(* CoDeSys 2.3.9.28 project: Automacao_ProjetoSemestral.pro *)
(* Libraries: Standard.lib 27.1.09 11:27:38, Util.lib 27.1.09 11:27:38, IecSfc.lib 24.11.08 08:07:15, SysLibTime.lib 27.1.09 11:27:38, SysTaskInfo.lib 24.11.08 08:07:15, SYSLIBCALLBACK.LIB 27.1.09 11:27:38 *)

(* PLC configuration (modules and I/O channels)
CPX-CEC [Root] node -1, in %IB0 out %QB0 {StringParam = 2773,0,0,0,0; ByteParam = 0; ByteParam = 31; ByteParam = 0; ByteParam = 0; ByteParam = 0; ByteParam = 0; ByteParam = 0; ByteParam = 0; ByteParam = 2; ByteParam = 0; ByteParam = 0; ByteParam = 0; ByteParam = 32; ByteParam = 0; ByteParam = 0; ByteParam = 5; ByteParam = 0; ByteParam = 0; ByteParam = 0; ByteParam = 0; ByteParam = 0; ByteParam = 0; ByteParam = 0; ByteParam = 0; ByteParam = 14; ByteParam = 240; ByteParam = 192; ByteParam = 168; ByteParam = 2; ByteParam = 10; ByteParam = 255; ByteParam = 255; ByteParam = 0; ByteParam = 0; ByteParam = 192; ByteParam = 168; ByteParam = 1; ByteParam = 1; ByteParam = 192; ByteParam = 168; ByteParam = 2; ByteParam = 10; ByteParam = 255; ByteParam = 255; ByteParam = 0; ByteParam = 0; ByteParam = 192; ByteParam = 168; ByteParam = 1; ByteParam = 1}
  Hexswitch AT %IB0 [HexSwitch] rotary switch 0 = STOP, 1-15 = RUN
  IOModules [CPX_MASTER] node 0, in %IB4 out %QB0
*)

(* Global variable list: Global_Variables *)
VAR_GLOBAL

	M1 : BOOL;
	M2 : BOOL;
	P1 : BOOL;
	P2_IDA : BOOL;
	P2_VOLTA : BOOL;
	P3 : BOOL;
	LP_1 : BOOL;
	LP_2 : BOOL;
	AL: BOOL;

	START AT %QX2.0 : BOOL;
	STOP AT %QX2.1 : BOOL;
	S1 AT %QX0.2 : BOOL;
	S2 AT %QX0.3 : BOOL;
	S3 AT %QX0.4 : BOOL;
	S4 AT %QX0.5 : BOOL;
	S5 AT %QX0.6 : BOOL;
	S6 AT %QX0.7 : BOOL;
	S7 AT %QX0.8 : BOOL;

	M_START : BOOL;
	M_CONT: BOOL;
	M_P1: BOOL;
	M_TEMPERA: BOOL;
	M_2_ENT : BOOL;
	M_2_SAI : BOOL;

	MT_1 : BOOL;
	MT_2 : BOOL;
	MT_3 : BOOL;
	MT_4 : BOOL;
	MT_5 : BOOL;

	T_TEMPERA : TON;
	T_P1 : TOF;
	T_ALARME1:TON;
	T_ALARME2:TON;

    CONT_2_ENT: CTU;
	CONT_2_SAI : CTU;

END_VAR

(* POU PLC_PRG, LD *)
PROGRAM PLC_PRG
VAR
END_VAR
VAR (* helpers for the ST form of the networks *)
	_p1 : BOOL;
	_p2 : BOOL;
	_p3 : BOOL;
END_VAR
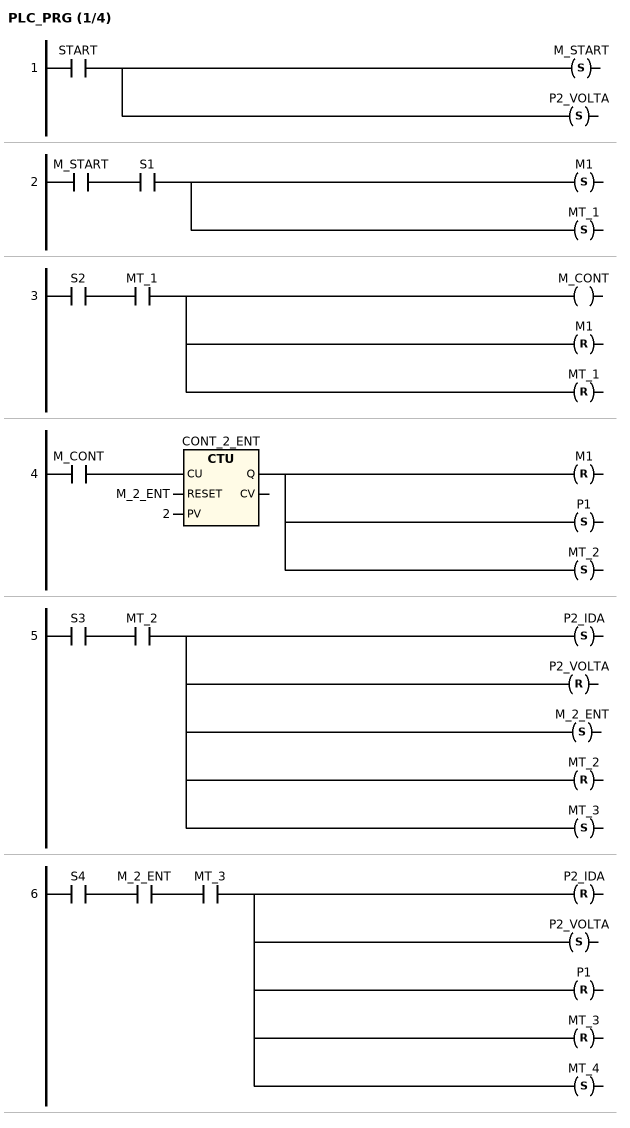
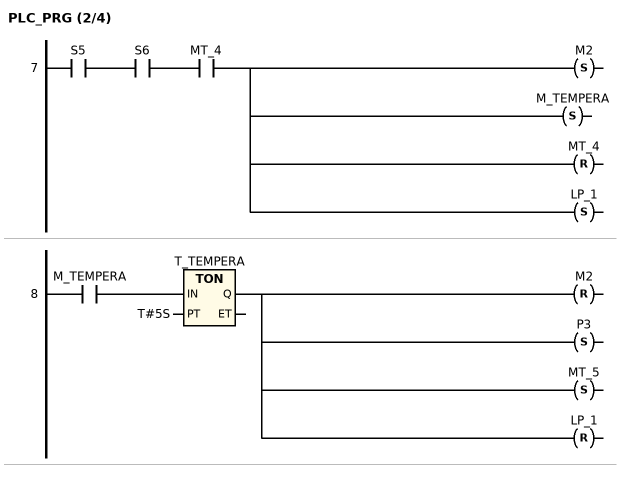
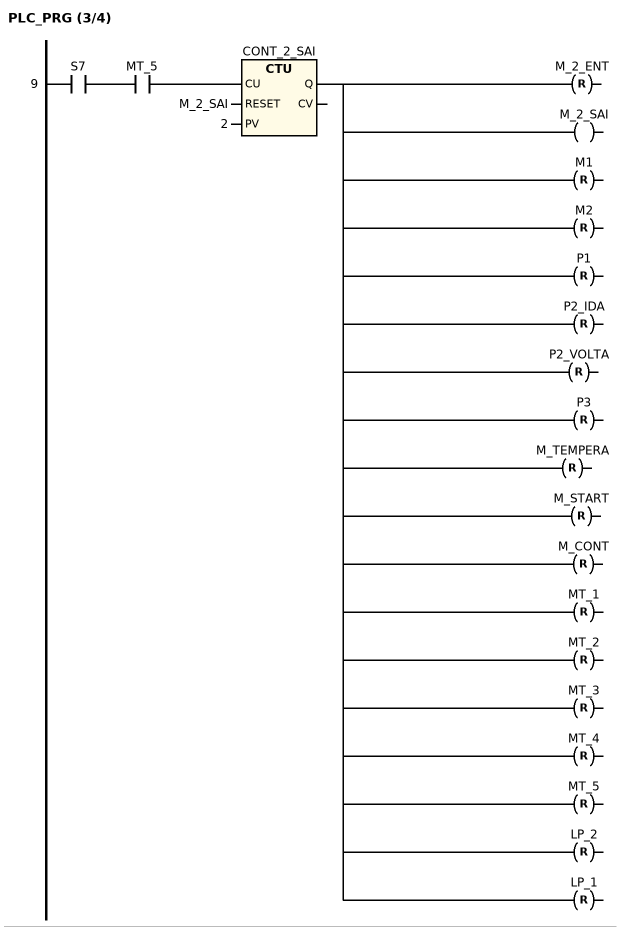
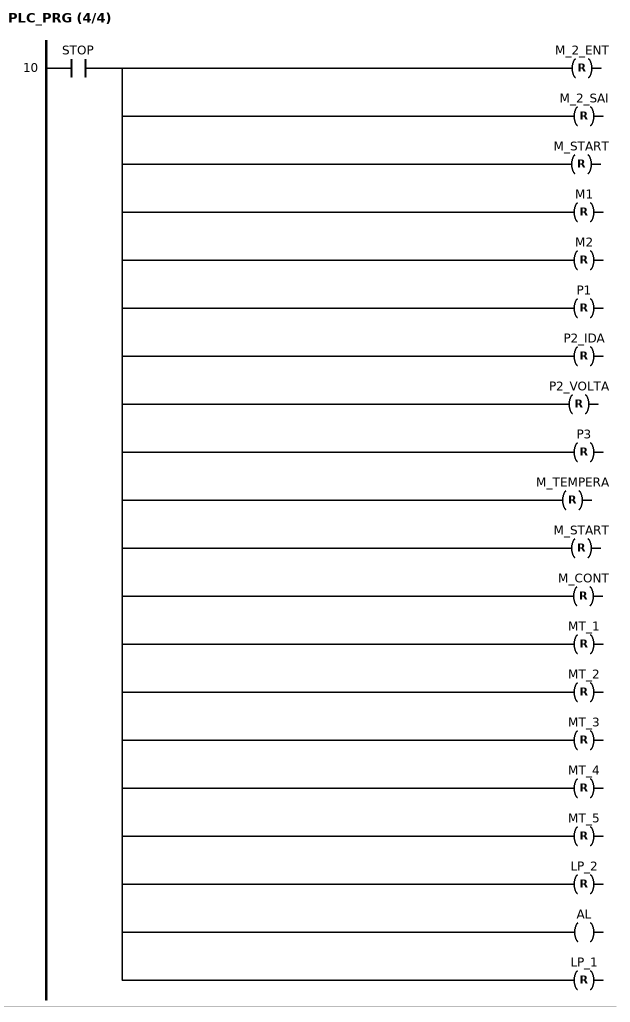
_LD_ (* Ladder Diagram *)
NETWORK 1
	[START] --- (S M_START) (S P2_VOLTA)
NETWORK 2
	[M_START] - [S1] --- (S M1) (S MT_1)
NETWORK 3
	[S2] - [MT_1] --- (M_CONT) (R M1) (R MT_1)
NETWORK 4
	[M_CONT] - CONT_2_ENT:CTU(CU: *, RESET: M_2_ENT, PV: 2) --- (R M1) (S P1) (S MT_2)
NETWORK 5
	[S3] - [MT_2] --- (S P2_IDA) (R P2_VOLTA) (S M_2_ENT) (R MT_2) (S MT_3)
NETWORK 6
	[S4] - [M_2_ENT] - [MT_3] --- (R P2_IDA) (S P2_VOLTA) (R P1) (R MT_3) (S MT_4)
NETWORK 7
	[S5] - [S6] - [MT_4] --- (S M2) (S M_TEMPERA) (R MT_4) (S LP_1)
NETWORK 8
	[M_TEMPERA] - T_TEMPERA:TON(IN: *, PT: T#5S) --- (R M2) (S P3) (S MT_5) (R LP_1)
NETWORK 9
	[S7] - [MT_5] - CONT_2_SAI:CTU(CU: *, RESET: M_2_SAI, PV: 2) --- (R M_2_ENT) (M_2_SAI) (R M1) (R M2) (R P1) (R P2_IDA) (R P2_VOLTA) (R P3) (R M_TEMPERA) (R M_START) (R M_CONT) (R MT_1) (R MT_2) (R MT_3) (R MT_4) (R MT_5) (R LP_2) (R LP_1)
NETWORK 10
	[STOP] --- (R M_2_ENT) (R M_2_SAI) (R M_START) (R M1) (R M2) (R P1) (R P2_IDA) (R P2_VOLTA) (R P3) (R M_TEMPERA) (R M_START) (R M_CONT) (R MT_1) (R MT_2) (R MT_3) (R MT_4) (R MT_5) (R LP_2) (AL) (R LP_1)
_END_LD_
(* the same logic as Structured Text *)
(* Network 1 *)
IF START THEN M_START := TRUE; P2_VOLTA := TRUE; END_IF;
(* Network 2 *)
IF M_START AND S1 THEN M1 := TRUE; MT_1 := TRUE; END_IF;
(* Network 3 *)
M_CONT := S2 AND MT_1;
IF M_CONT THEN M1 := FALSE; MT_1 := FALSE; END_IF;
(* Network 4 *)
CONT_2_ENT(CU := M_CONT, RESET := M_2_ENT, PV := 2);
IF CONT_2_ENT.Q THEN M1 := FALSE; P1 := TRUE; MT_2 := TRUE; END_IF;
(* Network 5 *)
_p1 := S3 AND MT_2;
IF _p1 THEN P2_IDA := TRUE; P2_VOLTA := FALSE; M_2_ENT := TRUE; MT_2 := FALSE; MT_3 := TRUE; END_IF;
(* Network 6 *)
_p2 := S4 AND M_2_ENT AND MT_3;
IF _p2 THEN P2_IDA := FALSE; P2_VOLTA := TRUE; P1 := FALSE; MT_3 := FALSE; MT_4 := TRUE; END_IF;
(* Network 7 *)
_p3 := S5 AND S6 AND MT_4;
IF _p3 THEN M2 := TRUE; M_TEMPERA := TRUE; MT_4 := FALSE; LP_1 := TRUE; END_IF;
(* Network 8 *)
T_TEMPERA(IN := M_TEMPERA, PT := T#5S);
IF T_TEMPERA.Q THEN M2 := FALSE; P3 := TRUE; MT_5 := TRUE; LP_1 := FALSE; END_IF;
(* Network 9 *)
CONT_2_SAI(CU := S7 AND MT_5, RESET := M_2_SAI, PV := 2);
IF CONT_2_SAI.Q THEN M_2_ENT := FALSE; END_IF;
M_2_SAI := CONT_2_SAI.Q;
IF CONT_2_SAI.Q THEN M1 := FALSE; END_IF;
IF CONT_2_SAI.Q THEN M2 := FALSE; END_IF;
IF CONT_2_SAI.Q THEN P1 := FALSE; END_IF;
IF CONT_2_SAI.Q THEN P2_IDA := FALSE; END_IF;
IF CONT_2_SAI.Q THEN P2_VOLTA := FALSE; END_IF;
IF CONT_2_SAI.Q THEN P3 := FALSE; END_IF;
IF CONT_2_SAI.Q THEN M_TEMPERA := FALSE; END_IF;
IF CONT_2_SAI.Q THEN M_START := FALSE; END_IF;
IF CONT_2_SAI.Q THEN M_CONT := FALSE; END_IF;
IF CONT_2_SAI.Q THEN MT_1 := FALSE; END_IF;
IF CONT_2_SAI.Q THEN MT_2 := FALSE; END_IF;
IF CONT_2_SAI.Q THEN MT_3 := FALSE; END_IF;
IF CONT_2_SAI.Q THEN MT_4 := FALSE; END_IF;
IF CONT_2_SAI.Q THEN MT_5 := FALSE; END_IF;
IF CONT_2_SAI.Q THEN LP_2 := FALSE; END_IF;
IF CONT_2_SAI.Q THEN LP_1 := FALSE; END_IF;
(* Network 10 *)
IF STOP THEN M_2_ENT := FALSE; END_IF;
IF STOP THEN M_2_SAI := FALSE; END_IF;
IF STOP THEN M_START := FALSE; END_IF;
IF STOP THEN M1 := FALSE; END_IF;
IF STOP THEN M2 := FALSE; END_IF;
IF STOP THEN P1 := FALSE; END_IF;
IF STOP THEN P2_IDA := FALSE; END_IF;
IF STOP THEN P2_VOLTA := FALSE; END_IF;
IF STOP THEN P3 := FALSE; END_IF;
IF STOP THEN M_TEMPERA := FALSE; END_IF;
IF STOP THEN M_START := FALSE; END_IF;
IF STOP THEN M_CONT := FALSE; END_IF;
IF STOP THEN MT_1 := FALSE; END_IF;
IF STOP THEN MT_2 := FALSE; END_IF;
IF STOP THEN MT_3 := FALSE; END_IF;
IF STOP THEN MT_4 := FALSE; END_IF;
IF STOP THEN MT_5 := FALSE; END_IF;
IF STOP THEN LP_2 := FALSE; END_IF;
AL := STOP;
IF STOP THEN LP_1 := FALSE; END_IF;
END_PROGRAM

(* Visualisation Simulacao
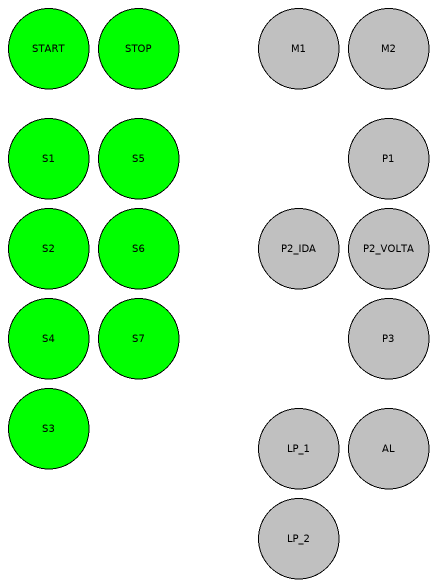
ellipse at (50,20)-(131,101): text "START"; alarm colour if START; taps START
ellipse at (140,20)-(221,101): text "STOP"; alarm colour if STOP; toggles STOP
ellipse at (50,130)-(131,211): text "S1"; alarm colour if S1; taps S1
ellipse at (50,220)-(131,301): text "S2"; alarm colour if S2; taps S2
ellipse at (50,400)-(131,481): text "S3"; alarm colour if S3; taps S3
ellipse at (50,310)-(131,391): text "S4"; alarm colour if S4; taps S4
ellipse at (140,130)-(221,211): text "S5"; alarm colour if S5; toggles S5
ellipse at (140,220)-(221,301): text "S6"; alarm colour if S6; taps S6
ellipse at (300,20)-(381,101): text "M1"; alarm colour if M1
ellipse at (390,20)-(471,101): text "M2"; alarm colour if M2
ellipse at (390,130)-(471,211): text "P1"; alarm colour if P1
ellipse at (390,220)-(471,301): text "P2_VOLTA"; alarm colour if P2_VOLTA
ellipse at (390,310)-(471,391): text "P3"; alarm colour if P3
ellipse at (300,220)-(381,301): text "P2_IDA"; alarm colour if P2_IDA
ellipse at (140,310)-(221,391): text "S7"; alarm colour if S7; taps S7
ellipse at (390,420)-(471,501): text "AL"; alarm colour if AL
ellipse at (300,420)-(381,501): text "LP_1"; alarm colour if LP_1
ellipse at (300,510)-(381,591): text "LP_2"; alarm colour if LP_2
*)
